// TIA Portal V16 export
// export: Created 2024-12-03T15:41:39.6418962Z, ExportSetting WithDefaults, DisplayName Totally Integrated Automation Portal, DisplayVersion V16 Update 6, DisplayName TIA Portal Version Control Interface, DisplayVersion V16 Update 2, DisplayName TIA Portal Openness, DisplayVersion V16 Update 6, DisplayName TIA Portal Teamcenter Gateway, DisplayVersion V16, DisplayName SINAMICS Startdrive Advanced, DisplayVersion V16 Update 5, DisplayName SINAMICS Startdrive G130, G150, S120, S150, SINAMICS MV, S210, DisplayVersion V16 Update 5, DisplayName SINAMICS Startdrive G110M, G120, G120C, G120D, G120P, G115D, DisplayVersion V16 Update 5, DisplayName STEP 7 Professional, DisplayVersion V16 Update 6, DisplayName STEP 7 Safety, DisplayVersion V16, DisplayName WinCC Advanced / Unified PC, DisplayVersion V16 Update 6
FUNCTION_BLOCK "CLX_FB"   // FB1, SCL
{ S7_Optimized_Access := 'TRUE' }
VERSION : 0.1
// stored: AutoNumber true, IsIECCheckEnabled false, IsRetainMemResEnabled false, MemoryReserve 100, SetENOAutomatically false, UDAEnableTagReadback false
   VAR
      MOT_102L : "ConveyLinxController_FullPLC";
      MOT_102R : "ConveyLinxController_FullPLC";
      MOT_103L : "ConveyLinxController_FullPLC";
      MOT_103R : "ConveyLinxController_FullPLC";
      MOT_104L : "ConveyLinxController_FullPLC";
      MOT_104R : "ConveyLinxController_FullPLC";
      MOT_105L : "ConveyLinxController_FullPLC";
      MOT_105R : "ConveyLinxController_FullPLC";
      MOT_106L : "ConveyLinxController_FullPLC";
      MOT_106R : "ConveyLinxController_FullPLC";
      MOT_107L : "FlowSort_Twister_Controller_FB";
      MOT_107R : "ConveyLinxController_FullPLC";
      MOT_108L : "ConveyLinxController_FullPLC";
      MOT_108R : "ConveyLinxController_FullPLC";
      MOT_109L : "ConveyLinxController_FullPLC";
      MOT_109R : "ConveyLinxController_FullPLC";
      MOT_110L : "ConveyLinxController_FullPLC";
      MOT_110R : "ConveyLinxController_FullPLC";
      MOT_111L : "ConveyLinxController_FullPLC";
      MOT_111R : "ConveyLinxController_FullPLC";
      MOT_112L : "ConveyLinxController_FullPLC";
      MOT_112R : "ConveyLinxController_FullPLC";
      MOT_113L : "ConveyLinxController_FullPLC";
      MOT_113R : "ConveyLinxController_FullPLC";
      MOT_114L : "ConveyLinxController_FullPLC";
      MOT_114R : "ConveyLinxController_FullPLC";
      MOT_115L : "ConveyLinxController_FullPLC";
      MOT_115R : "ConveyLinxController_FullPLC";
      MOT_201L { S7_SetPoint := 'True'} : "ES_TransferUnit_UpDown_Controller_Servo_FB";
      MOT_201R { S7_SetPoint := 'True'} : "ConveyLinxController_FullPLC";
      MOT_202L : "ConveyLinxController_FullPLC";
      MOT_202R : "ConveyLinxController_FullPLC";
      MOT_203L { S7_SetPoint := 'True'} : "ES_TransferUnit_UpDown_Controller_Servo_FB";
      MOT_203R : "ConveyLinxController_FullPLC";
      MOT_301L : "ConveyLinxController_FullPLC";
      MOT_301R : "ConveyLinxController_FullPLC";
      MOT_302L : "ConveyLinxController_FullPLC";
      MOT_302R : "ConveyLinxController_FullPLC";
      MOT_303L : "ConveyLinxController_FullPLC";
      MOT_303R : "ConveyLinxController_FullPLC";
      MOT_304L : "ConveyLinxController_FullPLC";
      MOT_304R : "ConveyLinxController_FullPLC";
      MOT_305L : "ConveyLinxController_FullPLC";
      MOT_305R : "ConveyLinxController_FullPLC";
   END_VAR
BEGIN

   REGION MOT_102L

       "Conv_Conveylinx_Commander"(I_INV := FALSE,
                                   I_Conv := "CONV_DB".CONV_102L,
                                   IO_ConveyLinxFullPLC := "MOT_CLX_DB".MOT_102L);

       #MOT_102L(I_MotorData := "I_CON_102",
                 I_ControlLeftMotorConveyLInx := TRUE,
                 I_ControlRightMotorConveyLinx := FALSE,
                 IO_MotorStatus := "MOT_CLX_DB".MOT_102L,
                 IO_MotorOutput := "Q_CON_102");

   END_REGION

   REGION MOT_102R

       "Conv_Conveylinx_Commander"(I_INV := FALSE,
                                   I_Conv := "CONV_DB".CONV_102R,
                                   IO_ConveyLinxFullPLC := "MOT_CLX_DB".MOT_102R);

       #MOT_102R(I_MotorData := "I_CON_102",
                 I_ControlLeftMotorConveyLInx := FALSE,
                 I_ControlRightMotorConveyLinx := TRUE,
                 IO_MotorStatus := "MOT_CLX_DB".MOT_102R,
                 IO_MotorOutput := "Q_CON_102");

   END_REGION

   REGION MOT_103L

       "Conv_Conveylinx_Commander"(I_INV := FALSE,
                                   I_Conv := "CONV_DB".CONV_103L,
                                   IO_ConveyLinxFullPLC := "MOT_CLX_DB".MOT_103L);

       #MOT_103L(I_MotorData := "I_CON_103",
                 I_ControlLeftMotorConveyLInx := TRUE,
                 I_ControlRightMotorConveyLinx := FALSE,
                 IO_MotorStatus := "MOT_CLX_DB".MOT_103L,
                 IO_MotorOutput := "Q_CON_103");

   END_REGION

   REGION MOT_103R

       "Conv_Conveylinx_Commander"(I_INV := FALSE,
                                   I_Conv := "CONV_DB".CONV_103R,
                                   IO_ConveyLinxFullPLC := "MOT_CLX_DB".MOT_103R);

       #MOT_103R(I_MotorData := "I_CON_103",
                 I_ControlLeftMotorConveyLInx := FALSE,
                 I_ControlRightMotorConveyLinx := TRUE,
                 IO_MotorStatus := "MOT_CLX_DB".MOT_103R,
                 IO_MotorOutput := "Q_CON_103");

   END_REGION

   REGION MOT_104L

       "Conv_Conveylinx_Commander"(I_INV := FALSE,
                                   I_Conv := "CONV_DB".CONV_104L,
                                   IO_ConveyLinxFullPLC := "MOT_CLX_DB".MOT_104L);

       #MOT_104L(I_MotorData := "I_CON_104",
                 I_ControlLeftMotorConveyLInx := TRUE,
                 I_ControlRightMotorConveyLinx := FALSE,
                 IO_MotorStatus := "MOT_CLX_DB".MOT_104L,
                 IO_MotorOutput := "Q_CON_104");

   END_REGION

   REGION MOT_104R

       "Conv_Conveylinx_Commander"(I_INV := FALSE,
                                   I_Conv := "CONV_DB".CONV_104R,
                                   IO_ConveyLinxFullPLC := "MOT_CLX_DB".MOT_104R);

       #MOT_104R(I_MotorData := "I_CON_104",
                 I_ControlLeftMotorConveyLInx := FALSE,
                 I_ControlRightMotorConveyLinx := TRUE,
                 IO_MotorStatus := "MOT_CLX_DB".MOT_104R,
                 IO_MotorOutput := "Q_CON_104");

   END_REGION

   REGION MOT_105L

       "Conv_Conveylinx_Commander"(I_INV := FALSE,
                                   I_Conv := "CONV_DB".CONV_105L,
                                   IO_ConveyLinxFullPLC := "MOT_CLX_DB".MOT_105L);

       #MOT_105L(I_MotorData := "I_CON_105",
                 I_ControlLeftMotorConveyLInx := TRUE,
                 I_ControlRightMotorConveyLinx := FALSE,
                 IO_MotorStatus := "MOT_CLX_DB".MOT_105L,
                 IO_MotorOutput := "Q_CON_105");

   END_REGION

   REGION MOT_105R

       "Conv_Conveylinx_Commander"(I_INV := FALSE,
                                   I_Conv := "CONV_DB".CONV_105R,
                                   IO_ConveyLinxFullPLC := "MOT_CLX_DB".MOT_105R);

       #MOT_105R(I_MotorData := "I_CON_105",
                 I_ControlLeftMotorConveyLInx := FALSE,
                 I_ControlRightMotorConveyLinx := TRUE,
                 IO_MotorStatus := "MOT_CLX_DB".MOT_105R,
                 IO_MotorOutput := "Q_CON_105");

   END_REGION

   REGION MOT_106L

       "Conv_Conveylinx_Commander"(I_INV := FALSE,
                                   I_Conv := "CONV_DB".CONV_107R,
                                   IO_ConveyLinxFullPLC := "MOT_CLX_DB".MOT_106L);

       #MOT_106L(I_MotorData := "I_CON_106",
                 I_ControlLeftMotorConveyLInx := TRUE,
                 I_ControlRightMotorConveyLinx := FALSE,
                 IO_MotorStatus := "MOT_CLX_DB".MOT_106L,
                 IO_MotorOutput := "Q_CON_106");

   END_REGION

   REGION MOT_106R

       "Conv_Conveylinx_Commander"(I_INV := FALSE,
                                   I_Conv := "CONV_DB".CONV_106R,
                                   IO_ConveyLinxFullPLC := "MOT_CLX_DB".MOT_106R);

       #MOT_106R(I_MotorData := "I_CON_106",
                 I_ControlLeftMotorConveyLInx := FALSE,
                 I_ControlRightMotorConveyLinx := TRUE,
                 IO_MotorStatus := "MOT_CLX_DB".MOT_106R,
                 IO_MotorOutput := "Q_CON_106");

   END_REGION

   REGION MOT_107L FLOWSORT


       #MOT_107L(I_MotorData := "I_CON_107",
                 I_ControlLeftMotorConveyLInx := TRUE,
                 I_ControlRightMotorConveyLinx := FALSE,
                 I_homeFeedback:="Inputs_DB".FTC_107_L4,
                 IO_MotorStatus := "MOT_CLX_DB".MOT_107L,
                 IO_MotorOutput := "Q_CON_107");


   END_REGION

   REGION MOT_107R

       "Conv_Conveylinx_Commander"(I_INV := FALSE,
                                   I_Conv := "CONV_DB".CONV_107R,
                                   IO_ConveyLinxFullPLC := "MOT_CLX_DB".MOT_107R);

       #MOT_107R(I_MotorData := "I_CON_107",
                 I_ControlLeftMotorConveyLInx := FALSE,
                 I_ControlRightMotorConveyLinx := TRUE,
                 IO_MotorStatus := "MOT_CLX_DB".MOT_107R,
                 IO_MotorOutput := "Q_CON_107");

   END_REGION

   REGION MOT_108L

       "Conv_Conveylinx_Commander"(I_INV := FALSE,
                                   I_Conv := "CONV_DB".CONV_108L,
                                   IO_ConveyLinxFullPLC := "MOT_CLX_DB".MOT_108L);

       #MOT_108L(I_MotorData := "I_CON_108",
                 I_ControlLeftMotorConveyLInx := TRUE,
                 I_ControlRightMotorConveyLinx := FALSE,
                 IO_MotorStatus := "MOT_CLX_DB".MOT_108L,
                 IO_MotorOutput := "Q_CON_108");

   END_REGION

   REGION MOT_108R

       "Conv_Conveylinx_Commander"(I_INV := FALSE,
                                   I_Conv := "CONV_DB".CONV_108R,
                                   IO_ConveyLinxFullPLC := "MOT_CLX_DB".MOT_108R);

       #MOT_108R(I_MotorData := "I_CON_108",
                 I_ControlLeftMotorConveyLInx := FALSE,
                 I_ControlRightMotorConveyLinx := TRUE,
                 IO_MotorStatus := "MOT_CLX_DB".MOT_108R,
                 IO_MotorOutput := "Q_CON_108");

   END_REGION

   REGION MOT_109L

       "Conv_Conveylinx_Commander"(I_INV := FALSE,
                                   I_Conv := "CONV_DB".CONV_109L,
                                   IO_ConveyLinxFullPLC := "MOT_CLX_DB".MOT_109L);

       #MOT_109L(I_MotorData := "I_CON_109",
                 I_ControlLeftMotorConveyLInx := TRUE,
                 I_ControlRightMotorConveyLinx := FALSE,
                 IO_MotorStatus := "MOT_CLX_DB".MOT_109L,
                 IO_MotorOutput := "Q_CON_109");

   END_REGION

   REGION MOT_109R

       "Conv_Conveylinx_Commander"(I_INV := FALSE,
                                   I_Conv := "CONV_DB".CONV_109R,
                                   IO_ConveyLinxFullPLC := "MOT_CLX_DB".MOT_109R);

       #MOT_109R(I_MotorData := "I_CON_109",
                 I_ControlLeftMotorConveyLInx := FALSE,
                 I_ControlRightMotorConveyLinx := TRUE,
                 IO_MotorStatus := "MOT_CLX_DB".MOT_109R,
                 IO_MotorOutput := "Q_CON_109");

   END_REGION

   REGION MOT_110L

       "Conv_Conveylinx_Commander"(I_INV := FALSE,
                                   I_Conv := "CONV_DB".CONV_110L,
                                   IO_ConveyLinxFullPLC := "MOT_CLX_DB".MOT_110L);

       #MOT_110L(I_MotorData := "I_CON_110",
                 I_ControlLeftMotorConveyLInx := TRUE,
                 I_ControlRightMotorConveyLinx := FALSE,
                 IO_MotorStatus := "MOT_CLX_DB".MOT_110L,
                 IO_MotorOutput := "Q_CON_110");

   END_REGION

   REGION MOT_110R

       "Conv_Conveylinx_Commander"(I_INV := FALSE,
                                   I_Conv := "CONV_DB".CONV_110R,
                                   IO_ConveyLinxFullPLC := "MOT_CLX_DB".MOT_110R);

       #MOT_110R(I_MotorData := "I_CON_110",
                 I_ControlLeftMotorConveyLInx := FALSE,
                 I_ControlRightMotorConveyLinx := TRUE,
                 IO_MotorStatus := "MOT_CLX_DB".MOT_110R,
                 IO_MotorOutput := "Q_CON_110");

   END_REGION

   REGION MOT_111L

       "Conv_Conveylinx_Commander"(I_INV := FALSE,
                                   I_Conv := "CONV_DB".CONV_111L,
                                   IO_ConveyLinxFullPLC := "MOT_CLX_DB".MOT_111L);

       #MOT_111L(I_MotorData := "I_CON_111",
                 I_ControlLeftMotorConveyLInx := TRUE,
                 I_ControlRightMotorConveyLinx := FALSE,
                 IO_MotorStatus := "MOT_CLX_DB".MOT_111L,
                 IO_MotorOutput := "Q_CON_111");

   END_REGION

   REGION MOT_111R

       "Conv_Conveylinx_Commander"(I_INV := FALSE,
                                   I_Conv := "CONV_DB".CONV_111R,
                                   IO_ConveyLinxFullPLC := "MOT_CLX_DB".MOT_111R);

       #MOT_111R(I_MotorData := "I_CON_111",
                 I_ControlLeftMotorConveyLInx := FALSE,
                 I_ControlRightMotorConveyLinx := TRUE,
                 IO_MotorStatus := "MOT_CLX_DB".MOT_111R,
                 IO_MotorOutput := "Q_CON_111");

   END_REGION

   REGION MOT_112L

       "Conv_Conveylinx_Commander"(I_INV := FALSE,
                                   I_Conv := "CONV_DB".CONV_113L,
                                   IO_ConveyLinxFullPLC := "MOT_CLX_DB".MOT_112L);

       #MOT_112L(I_MotorData := "I_CON_112",
                 I_ControlLeftMotorConveyLInx := TRUE,
                 I_ControlRightMotorConveyLinx := FALSE,
                 IO_MotorStatus := "MOT_CLX_DB".MOT_112L,
                 IO_MotorOutput := "Q_CON_112");

   END_REGION

   REGION MOT_112R

       "Conv_Conveylinx_Commander"(I_INV := FALSE,
                                   I_Conv := "CONV_DB".CONV_112R,
                                   IO_ConveyLinxFullPLC := "MOT_CLX_DB".MOT_112R);

       #MOT_112R(I_MotorData := "I_CON_112",
                 I_ControlLeftMotorConveyLInx := FALSE,
                 I_ControlRightMotorConveyLinx := TRUE,
                 IO_MotorStatus := "MOT_CLX_DB".MOT_112R,
                 IO_MotorOutput := "Q_CON_112");

   END_REGION

   REGION MOT_113L

       "Conv_Conveylinx_Commander"(I_INV := FALSE,
                                   I_Conv := "CONV_DB".CONV_113L,
                                   IO_ConveyLinxFullPLC := "MOT_CLX_DB".MOT_113L);

       #MOT_113L(I_MotorData := "I_CON_113",
                 I_ControlLeftMotorConveyLInx := TRUE,
                 I_ControlRightMotorConveyLinx := FALSE,
                 IO_MotorStatus := "MOT_CLX_DB".MOT_113L,
                 IO_MotorOutput := "Q_CON_113");

   END_REGION

   REGION MOT_113R

       "Conv_Conveylinx_Commander"(I_INV := FALSE,
                                   I_Conv := "CONV_DB".CONV_113R,
                                   IO_ConveyLinxFullPLC := "MOT_CLX_DB".MOT_113R);

       #MOT_113R(I_MotorData := "I_CON_113",
                 I_ControlLeftMotorConveyLInx := FALSE,
                 I_ControlRightMotorConveyLinx := TRUE,
                 IO_MotorStatus := "MOT_CLX_DB".MOT_113R,
                 IO_MotorOutput := "Q_CON_113");

   END_REGION

   REGION MOT_114L

       "Conv_Conveylinx_Commander"(I_INV := FALSE,
                                   I_Conv := "CONV_DB".CONV_114L,
                                   IO_ConveyLinxFullPLC := "MOT_CLX_DB".MOT_114L);

       #MOT_114L(I_MotorData := "I_CON_114",
                 I_ControlLeftMotorConveyLInx := TRUE,
                 I_ControlRightMotorConveyLinx := FALSE,
                 IO_MotorStatus := "MOT_CLX_DB".MOT_114L,
                 IO_MotorOutput := "Q_CON_114");

   END_REGION

   REGION MOT_114R

       "Conv_Conveylinx_Commander"(I_INV := FALSE,
                                   I_Conv := "CONV_DB".CONV_114R,
                                   IO_ConveyLinxFullPLC := "MOT_CLX_DB".MOT_114R);

       #MOT_114R(I_MotorData := "I_CON_114",
                 I_ControlLeftMotorConveyLInx := FALSE,
                 I_ControlRightMotorConveyLinx := TRUE,
                 IO_MotorStatus := "MOT_CLX_DB".MOT_114R,
                 IO_MotorOutput := "Q_CON_114");

   END_REGION

   REGION MOT_115L

       "Conv_Conveylinx_Commander"(I_INV := FALSE,
                                   I_Conv := "CONV_DB".CONV_115L,
                                   IO_ConveyLinxFullPLC := "MOT_CLX_DB".MOT_115L);

       #MOT_115L(I_MotorData := "I_CON_115",
                 I_ControlLeftMotorConveyLInx := TRUE,
                 I_ControlRightMotorConveyLinx := FALSE,
                 IO_MotorStatus := "MOT_CLX_DB".MOT_115L,
                 IO_MotorOutput := "Q_CON_115");

   END_REGION

   REGION MOT_115R

       "Conv_Conveylinx_Commander"(I_INV := FALSE,
                                   I_Conv := "CONV_DB".CONV_115R,
                                   IO_ConveyLinxFullPLC := "MOT_CLX_DB".MOT_115R);

       #MOT_115R(I_MotorData := "I_CON_115",
                 I_ControlLeftMotorConveyLInx := FALSE,
                 I_ControlRightMotorConveyLinx := TRUE,
                 IO_MotorStatus := "MOT_CLX_DB".MOT_115R,
                 IO_MotorOutput := "Q_CON_115");

   END_REGION

   REGION MOT_201L

       "Transfer_UpDown_EasySystems_Transfer_Interface_FC"(IO_TransferLogic := "TRANSFER_DB".T201L,
                                                           IO_EasySystemsTransfer := "MOT_CLX_DB".MOT_201L_Lift);

       #MOT_201L(I_MotorData := "I_CON_201",
                 I_ControlLeftMotorConveyLInx := TRUE,
                 I_ControlRightMotorConveyLinx := FALSE,
                 I_UpFb := "Inputs_DB".FTC_201_L4,
                 IO_MotorStatus := "MOT_CLX_DB".MOT_201L_Lift,
                 IO_MotorOutput := "Q_CON_201");


   END_REGION

   REGION MOT_201R

       "Conv_Conveylinx_Commander"(I_INV := FALSE,
                                   I_Conv := "CONV_DB".CONV_201R_BELTS,
                                   IO_ConveyLinxFullPLC := "MOT_CLX_DB".MOT_201R_Belts);

       #MOT_201R(I_MotorData := "I_CON_201",
                 I_ControlLeftMotorConveyLInx := FALSE,
                 I_ControlRightMotorConveyLinx := TRUE,
                 IO_MotorStatus := "MOT_CLX_DB".MOT_201R_Belts,
                 IO_MotorOutput := "Q_CON_201");

   END_REGION

   REGION MOT_202L

       "Conv_Conveylinx_Commander"(I_INV := FALSE,
                                   I_Conv := "CONV_DB".CONV_203R_BELTS,
                                   IO_ConveyLinxFullPLC := "MOT_CLX_DB".MOT_202L);

       #MOT_202L(I_MotorData := "I_CON_202",
                 I_ControlLeftMotorConveyLInx := TRUE,
                 I_ControlRightMotorConveyLinx := FALSE,
                 IO_MotorStatus := "MOT_CLX_DB".MOT_202L,
                 IO_MotorOutput := "Q_CON_202");

   END_REGION

   REGION MOT_202R

       "Conv_Conveylinx_Commander"(I_INV := FALSE,
                                   I_Conv := "CONV_DB".CONV_203R_BELTS,
                                   IO_ConveyLinxFullPLC := "MOT_CLX_DB".MOT_202R);

       #MOT_202R(I_MotorData := "I_CON_202",
                 I_ControlLeftMotorConveyLInx := FALSE,
                 I_ControlRightMotorConveyLinx := TRUE,
                 IO_MotorStatus := "MOT_CLX_DB".MOT_202R,
                 IO_MotorOutput := "Q_CON_202");

   END_REGION

   REGION MOT_203L

       "Transfer_UpDown_EasySystems_Transfer_Interface_FC"(IO_TransferLogic:="TRANSFER_DB".T203L,
                                                           IO_EasySystemsTransfer:="MOT_CLX_DB".MOT_203L_Lift);

       #MOT_203L(I_MotorData := "I_CON_203",
                 I_ControlLeftMotorConveyLInx := TRUE,
                 I_ControlRightMotorConveyLinx := FALSE,
                 I_UpFb:="Inputs_DB".FTC_203_L4,
                 IO_MotorStatus := "MOT_CLX_DB".MOT_203L_Lift,
                 IO_MotorOutput := "Q_CON_203");


   END_REGION

   REGION MOT_203R

       "Conv_Conveylinx_Commander"(I_INV := FALSE,
                                   I_Conv := "CONV_DB".CONV_203R_BELTS,
                                   IO_ConveyLinxFullPLC := "MOT_CLX_DB".MOT_203R_Belts);

       #MOT_203R(I_MotorData := "I_CON_203",
                 I_ControlLeftMotorConveyLInx := FALSE,
                 I_ControlRightMotorConveyLinx := TRUE,
                 IO_MotorStatus := "MOT_CLX_DB".MOT_203R_Belts,
                 IO_MotorOutput := "Q_CON_203");

   END_REGION

   REGION MOT_301L

       "Conv_Conveylinx_Commander"(I_INV := FALSE,
                                   I_Conv := "CONV_DB".CONV_301R,
                                   IO_ConveyLinxFullPLC := "MOT_CLX_DB".MOT_301L);

       #MOT_301L(I_MotorData := "I_CON_301",
                 I_ControlLeftMotorConveyLInx := TRUE,
                 I_ControlRightMotorConveyLinx := FALSE,
                 IO_MotorStatus := "MOT_CLX_DB".MOT_301L,
                 IO_MotorOutput := "Q_CON_301");

   END_REGION

   REGION MOT_301R

       "Conv_Conveylinx_Commander"(I_INV := FALSE,
                                   I_Conv := "CONV_DB".CONV_301R,
                                   IO_ConveyLinxFullPLC := "MOT_CLX_DB".MOT_301R);

       #MOT_301R(I_MotorData := "I_CON_301",
                 I_ControlLeftMotorConveyLInx := FALSE,
                 I_ControlRightMotorConveyLinx := TRUE,
                 IO_MotorStatus := "MOT_CLX_DB".MOT_301R,
                 IO_MotorOutput := "Q_CON_301");

   END_REGION

   REGION MOT_302L

       "Conv_Conveylinx_Commander"(I_INV := FALSE,
                                   I_Conv := "CONV_DB".CONV_302L,
                                   IO_ConveyLinxFullPLC := "MOT_CLX_DB".MOT_302L);

       #MOT_302L(I_MotorData := "I_CON_302",
                 I_ControlLeftMotorConveyLInx := TRUE,
                 I_ControlRightMotorConveyLinx := FALSE,
                 IO_MotorStatus := "MOT_CLX_DB".MOT_302L,
                 IO_MotorOutput := "Q_CON_302");

   END_REGION

   REGION MOT_302R

       "Conv_Conveylinx_Commander"(I_INV := FALSE,
                                   I_Conv := "CONV_DB".CONV_302R,
                                   IO_ConveyLinxFullPLC := "MOT_CLX_DB".MOT_302R);

       #MOT_302R(I_MotorData := "I_CON_302",
                 I_ControlLeftMotorConveyLInx := FALSE,
                 I_ControlRightMotorConveyLinx := TRUE,
                 IO_MotorStatus := "MOT_CLX_DB".MOT_302R,
                 IO_MotorOutput := "Q_CON_302");

   END_REGION

   REGION MOT_303L

       "Conv_Conveylinx_Commander"(I_INV := FALSE,
                                   I_Conv := "CONV_DB".CONV_303L,
                                   IO_ConveyLinxFullPLC := "MOT_CLX_DB".MOT_303L);

       #MOT_303L(I_MotorData := "I_CON_303",
                 I_ControlLeftMotorConveyLInx := TRUE,
                 I_ControlRightMotorConveyLinx := FALSE,
                 IO_MotorStatus := "MOT_CLX_DB".MOT_303L,
                 IO_MotorOutput := "Q_CON_303");

   END_REGION

   REGION MOT_303R

       "Conv_Conveylinx_Commander"(I_INV := FALSE,
                                   I_Conv := "CONV_DB".CONV_303R,
                                   IO_ConveyLinxFullPLC := "MOT_CLX_DB".MOT_303R);

       #MOT_303R(I_MotorData := "I_CON_303",
                 I_ControlLeftMotorConveyLInx := FALSE,
                 I_ControlRightMotorConveyLinx := TRUE,
                 IO_MotorStatus := "MOT_CLX_DB".MOT_303R,
                 IO_MotorOutput := "Q_CON_303");

   END_REGION

   REGION MOT_304L

       "Conv_Conveylinx_Commander"(I_INV := FALSE,
                                   I_Conv := "CONV_DB".CONV_304L,
                                   IO_ConveyLinxFullPLC := "MOT_CLX_DB".MOT_304L);

       #MOT_304L(I_MotorData := "I_CON_304",
                 I_ControlLeftMotorConveyLInx := TRUE,
                 I_ControlRightMotorConveyLinx := FALSE,
                 IO_MotorStatus := "MOT_CLX_DB".MOT_304L,
                 IO_MotorOutput := "Q_CON_304");

   END_REGION

   REGION MOT_304R

       "Conv_Conveylinx_Commander"(I_INV := FALSE,
                                   I_Conv := "CONV_DB".CONV_304R,
                                   IO_ConveyLinxFullPLC := "MOT_CLX_DB".MOT_304R);

       #MOT_304R(I_MotorData := "I_CON_304",
                 I_ControlLeftMotorConveyLInx := FALSE,
                 I_ControlRightMotorConveyLinx := TRUE,
                 IO_MotorStatus := "MOT_CLX_DB".MOT_304R,
                 IO_MotorOutput := "Q_CON_304");

   END_REGION

   REGION MOT_305L

       "Conv_Conveylinx_Commander"(I_INV := FALSE,
                                   I_Conv := "CONV_DB".CONV_305R,
                                   IO_ConveyLinxFullPLC := "MOT_CLX_DB".MOT_305L);

       #MOT_305L(I_MotorData := "I_CON_305",
                 I_ControlLeftMotorConveyLInx := TRUE,
                 I_ControlRightMotorConveyLinx := FALSE,
                 IO_MotorStatus := "MOT_CLX_DB".MOT_305L,
                 IO_MotorOutput := "Q_CON_305");

   END_REGION

   REGION MOT_305R

       "Conv_Conveylinx_Commander"(I_INV := FALSE,
                                   I_Conv := "CONV_DB".CONV_305R,
                                   IO_ConveyLinxFullPLC := "MOT_CLX_DB".MOT_305R);

       #MOT_305R(I_MotorData := "I_CON_305",
                 I_ControlLeftMotorConveyLInx := FALSE,
                 I_ControlRightMotorConveyLinx := TRUE,
                 IO_MotorStatus := "MOT_CLX_DB".MOT_305R,
                 IO_MotorOutput := "Q_CON_305");

   END_REGION
END_FUNCTION_BLOCK
